PROGRAM MAIN
VAR
END_VAR

METHOD FB_init : BOOL
VAR_INPUT
	bInitRetains : BOOL; // if TRUE, the retain variables are initialized (warm start / cold start)
	bInCopyCode : BOOL;  // if TRUE, the instance afterwards gets moved into the copy code (online change)
END_VAR
END_METHOD

END_PROGRAM

(* stored: Version 1.1.0.1, ProductVersion 3.1.4024.12
   POU MAIN: Id {0e98ea23-83dd-4ca9-a69f-2f12044496e3}, SpecialFunc None
   Method FB_init: Id {7294592a-873a-4442-84ee-f4182895888d} *)
